// TIA Portal V19 export
DATA_BLOCK "SafetyDataExchangeDB"   // DB7
{ S7_Optimized_Access := 'TRUE' }
// stored: MemoryReserve 100
   VAR
      SubordinateClockByte : Int;
   END_VAR
BEGIN
END_DATA_BLOCK
